# B&R Automation Studio project develop (part 8)

### Package Logical/P84Sample - Sample for ACOPOSinverter P84

### Data object Logical/P84Sample/P84config (Simple) - Inverter- Parameter

#### P84config.dat
```
(********************************************************************
 * COPYRIGHT -- Bernecker + Rainer
 ********************************************************************
 * Author:
 * Created:
 ********************************************************************
 * Allgemeine Syntax:
 * "<Parametername> = <Wert>"   oder
 * "<Parametername> = <symbolische Konstante>
 * Werte sind als Dezimalzahlen einzugeben
 ********************************************************************)
"bFr = 50"		; Standard- Motorfrequenz [50/60]
"IPL = nO"		; Verlust Netzphase
"nPr = 18"		; Motornennleistung [* 10W]
"UnS = 400"		; Motornennspannung [V]
"nCr = 14"		; Motornennstrom [* 0.1 A]
"FrS = 500"		; Motornennfrequenz [* 0.1 Hz]
"nSP = 880"	    ; Motornenndrehzahl [1/min]
"tFr = 600"		; maximale Ausgangsfrequenz [* 0.1 Hz]
"tUn = YES"		; Motormessung [nO/YES]
"PHr = AbC"		; Phasendrehung [AbC/ACb]
"ItH = 12"		; Thermischer Motornennstrom [* 0.1A]
"ACC = 5"		; Sollwertrampe-Hochlaufzeit [s]
"dEC = 5"		; Sollwertrampe-Auslaufzeit [s]
"LSP = 0"		; Motorfrequenz mit minimalem Sollwert [* 0.1 Hz]
"HSP = 600"		; Motorfrequenz mit maximalem Sollwert [* 0.1 Hz]
```

### Program Logical/P84Sample/P84 (IEC) - sample for ACOPOSinverter P84

#### P84Cyclic.ab - Zyklischer Code
```automation-basic
PROGRAM _CYCLIC

ac_inv_0 FUB ac_inv()

END_PROGRAM
```

#### P84Init.ab - Initialisierungscode
```automation-basic
PROGRAM _INIT

	ac_inv_alloc_0.pDevice = "IF3.ST4" // X20CP3585 internal EPL-IF @ node 4
	//ac_inv_alloc_0.pDevice = "SS1.IF1.ST2" // CANopen	node 2
	ac_inv_alloc_0.pcfgpar[0] = "P84config"  ; configuration data module
	ac_inv_alloc_0 FUB ac_inv_alloc()
	ac_inv_0.ax_ident = ac_inv_alloc_0.ax_ident

END_PROGRAM
```

### Package Logical/P74Sample - Sample for ACOPOSinverter

### Data object Logical/P74Sample/P74config (Simple) - Inverter- Parameter

#### P74config.dat
```
(********************************************************************
 * COPYRIGHT -- Bernecker + Rainer
 ********************************************************************
 * Author:
 * Created:
 ********************************************************************
 * Allgemeine Syntax:
 * "<Parametername> = <Wert>"   oder
 * "<Parametername> = <symbolische Konstante>
 * Werte sind als Dezimalzahlen einzugeben
 ********************************************************************)
"bFr = 50"		; Standard- Motorfrequenz [50/60]
"IPL = nO"		; Verlust Netzphase ( nur bei 3ph- Umrichter )
"nPr = 18"		; Motornennleistung [* 10W]
"UnS = 230"		; Motornennspannung [V]
"nCr = 14"		; Motornennstrom [* 0.1 A]
"COS = 88"		; Cosinus Phi [0.01]
"FrS = 500"		; Motornennfrequenz [* 0.1 Hz]
"nSP = 880"	    ; Motornenndrehzahl [1/min]
"tFr = 600"		; maximale Ausgangsfrequenz [* 0.1 Hz]
"ItH = 14"		; Thermischer Motornennstrom [* 0.1A]
"ACC = 5"		; Sollwertrampe-Hochlaufzeit [s]
"dEC = 5"		; Sollwertrampe-Auslaufzeit [s]
"LSP = 0"		; Motorfrequenz mit minimalem Sollwert [* 0.1 Hz]
"HSP = 600"		; Motorfrequenz mit maximalem Sollwert [* 0.1 Hz]
"OPL = nO"		; test without motor connected
```

### Program Logical/P74Sample/P74 (IEC) - P74 - Sample

#### P74Init.st - Initialisierungscode
```iecst
PROGRAM _INIT

	ac_inv_alloc_0.pDevice := 	ADR('IF3.ST10');  			(* X20 CP3585 internal EPL @ node 10 *)
	ac_inv_alloc_0.pcfgpar[0] :=  ADR('P74config');	 	(* configuration data module *)
	ac_inv_alloc_0.rpm := TRUE;	  (* use rpm instead of Hertz *)
	ac_inv_alloc_0();
	ac_inv_0.ax_ident := ac_inv_alloc_0.ax_ident;

END_PROGRAM
```

#### P74.var - Lokale Variablen
```iecst
VAR
	debug : REFERENCE TO ac_inv_AxIdent;
	ac_inv_alloc_0 : ac_inv_alloc;
	ac_inv_0 : ac_inv;
END_VAR
```

### Program Logical/P66Sample/P66C (IEC) - P66 with CAN - Sample

#### P66CInit.st - Initialisierungscode
```iecst
PROGRAM _INIT

	ac_inv_alloc_0.pDevice := 	ADR('SS1.IF1.ST2');     (* X20IF2772 - node 2 *)
	ac_inv_alloc_0.pcfgpar[0] :=  ADR('P66config');	 	(* configuration data module *)
	ac_inv_alloc_0();
	ac_inv_0.ax_ident := ac_inv_alloc_0.ax_ident;
END_PROGRAM
```

#### P66CCyclic.st - Zyklischer Code
```iecst
PROGRAM _CYCLIC

	ac_inv_0();

	IF( ac_inv_0.initialized AND ac_inv_0.ctrl_ready ) THEN
		ac_inv_0.ctrl_on := TRUE;
		IF( ac_inv_0.ctrl_is_on )THEN
			ac_inv_0.n_set := 100;
		END_IF
	END_IF

END_PROGRAM
```

### Program Logical/P66Sample/P66 (IEC) - P66 - EPL- Sample

#### P66Cyclic.st - Zyklischer Code
```iecst
PROGRAM _CYCLIC

	ac_inv_0();

	IF( ac_inv_0.initialized AND ac_inv_0.ctrl_ready ) THEN
		ac_inv_0.ctrl_on := TRUE;
		IF( ac_inv_0.ctrl_is_on )THEN
			ac_inv_0.n_set := 100;
		END_IF
	END_IF

END_PROGRAM
```

#### P66Init.st - Initialisierungscode
```iecst
PROGRAM _INIT

	ac_inv_alloc_0.pDevice := 	ADR('IF3.ST11');  		(* X20 CP3585 internal EPL @ node 11 *)
	ac_inv_alloc_0.pcfgpar[0] :=  ADR('P66config');	 	(* configuration data module *)
	ac_inv_alloc_0();
	ac_inv_0.ax_ident := ac_inv_alloc_0.ax_ident;
END_PROGRAM
```

#### P66.var - Lokale Variablen
```iecst
VAR
	ac_inv_alloc_0 : ac_inv_alloc;
	ac_inv_0 : ac_inv;
END_VAR
```

### Program Logical/P76Sample/P76 (IEC) - P76 - EPL- Sample

#### P76Cyclic.st - Zyklischer Code
```iecst
PROGRAM _CYCLIC

	ac_inv_0();

	IF( ac_inv_0.initialized AND ac_inv_0.ctrl_ready ) THEN
		ac_inv_0.ctrl_on := TRUE;
		IF( ac_inv_0.ctrl_is_on )THEN
			ac_inv_0.n_set := 100;
		END_IF
	END_IF

END_PROGRAM
```

#### P76Init.st - Initialisierungscode
```iecst
PROGRAM _INIT

	ac_inv_alloc_0.pDevice := 	ADR('IF3.ST5');  		(* X20 CP3585 internal EPL @ node 5 *)
	ac_inv_alloc_0.pcfgpar[0] := ADR('P76config');	 	(* configuration data module *)
	ac_inv_alloc_0();
	ac_inv_0.ax_ident := ac_inv_alloc_0.ax_ident;
END_PROGRAM
```

### Program Logical/P76Sample/P76C (IEC) - P76 with CAN - Sample

#### P76CInit.st - Initialisierungscode
```iecst
PROGRAM _INIT

	ac_inv_alloc_0.pDevice := 	ADR('IF7.ST2');     (* X20BB57 - node 2 *)
	ac_inv_alloc_0.pcfgpar[0] :=  ADR('P76config');	 	(* configuration data module *)
	ac_inv_alloc_0();
	ac_inv_0.ax_ident := ac_inv_alloc_0.ax_ident;
END_PROGRAM
```

#### P76CCyclic.st - Zyklischer Code
```iecst
PROGRAM _CYCLIC

	ac_inv_0();

//	IF( ac_inv_0.initialized AND ac_inv_0.ctrl_ready ) THEN
//		ac_inv_0.ctrl_on := TRUE;
//		IF( ac_inv_0.ctrl_is_on )THEN
//			ac_inv_0.n_set := 10;
//		END_IF
//	END_IF

END_PROGRAM
```

### Program Logical/P86Sample/P86 (IEC) - P86- EPL- Sample

#### P86Cyclic.st
```iecst
PROGRAM _CYCLIC

	ac_inv_0();

	IF  ac_inv_0.initialized AND ac_inv_0.ctrl_ready THEN
		IF ctrl_on THEN
			ac_inv_0.ctrl_on := TRUE;
			IF run THEN
				IF ac_inv_0.ctrl_is_on THEN
					ac_inv_0.n_set := 5;
				END_IF
			END_IF
		END_IF
	END_IF
END_PROGRAM
```

#### P86Init.st
```iecst
PROGRAM _INIT

	ac_inv_alloc_0.pDevice := ADR('IF3.ST2'); // X20CP3585 internal EPL-IF @ node 4
	ac_inv_alloc_0;
	ac_inv_alloc_0.pcfgpar[0] := ADR('P86config'); // configuration data module
	ac_inv_alloc_0();
	ac_inv_0.ax_ident := ac_inv_alloc_0.ax_ident;

END_PROGRAM
```

#### P86.var
```iecst
VAR
	ctrl_on : BOOL := FALSE;
	run : BOOL := FALSE;
	ac_inv_alloc_0 : ac_inv_alloc;
	ac_inv_0 : ac_inv;
END_VAR
```

#### P86Cyclic.ab - not listed in the package file held
```automation-basic
PROGRAM _CYCLIC

	ac_inv_0 FUB ac_inv()

	IF( ac_inv_0.initialized AND ac_inv_0.ctrl_ready ) THEN
		IF ctrl_on THEN

			ac_inv_0.ctrl_on := TRUE;
			IF run THEN

				IF( ac_inv_0.ctrl_is_on )THEN
					ac_inv_0.n_set := 5;
				ENDIF
			ENDIF
		ENDIF
	ENDIF

END_PROGRAM
```

#### P86Init.ab - not listed in the package file held
```automation-basic
PROGRAM _INIT

	ac_inv_alloc_0.pDevice = "IF3.ST2" // X20CP3585 internal EPL-IF @ node 4
	ac_inv_alloc_0
	//ac_inv_alloc_0.pDevice = "SS1.IF1.ST2" // CANopen	node 2
	ac_inv_alloc_0.pcfgpar[0] = "P86config"  ; configuration data module
	ac_inv_alloc_0 FUB ac_inv_alloc()
	ac_inv_0.ax_ident = ac_inv_alloc_0.ax_ident

END_PROGRAM
```

### Program Logical/P86Sample/P86_4_5 (IEC) - P86 size 4-5 - Sample

#### P86Init.ab - Initialisierungscode
```automation-basic
PROGRAM _INIT

	ac_inv_alloc_0.pDevice = "IF3.ST3" // X20CP3585 internal EPL-IF @ node 4
	//ac_inv_alloc_0.pDevice = "SS1.IF1.ST2" // CANopen	node 2
	ac_inv_alloc_0.pcfgpar[0] = "P86config4"  ; configuration data module
	ac_inv_alloc_0 FUB ac_inv_alloc()
	ac_inv_0.ax_ident = ac_inv_alloc_0.ax_ident

END_PROGRAM
```

#### P86Cyclic.st - not listed in the package file held
```iecst
PROGRAM _CYCLIC

	ac_inv_0();

	IF ac_inv_0.initialized AND ac_inv_0.ctrl_ready THEN
		IF ctrl_on THEN
			ac_inv_0.ctrl_on := TRUE;
			IF run THEN
				IF ac_inv_0.ctrl_is_on THEN
					ac_inv_0.n_set := 5;
				END_IF
			END_IF
		END_IF
	END_IF

END_PROGRAM
```

#### P86Init.st - not listed in the package file held
```iecst
PROGRAM _INIT

	ac_inv_alloc_0.pDevice := ADR('IF3.ST3'); // X20CP3585 internal EPL-IF @ node 4
	ac_inv_alloc_0.pcfgpar[0] := ADR('P86config4'); // configuration data module
	ac_inv_alloc_0();
	ac_inv_0.ax_ident := ac_inv_alloc_0.ax_ident;

END_PROGRAM
```

Listed in the project but not available here: Logical/P84Sample/P84/P84.var, Logical/P74Sample/P74/P74Cyclic.st, Logical/P66Sample/P66C/P66C.var, Logical/P76Sample/P76/P76.var, Logical/P76Sample/P76C/P76C.var, Logical/P86Sample/P86_4_5/P86Cyclic.ab, Logical/P86Sample/P86_4_5/P86.var
